SUBAPPLICATION GreenWhiteBackground3_AXSC (* Hintergrundfarbe (TRUE -> Grün, FALSE -> Weiß) für 3 Objekte (AX-Adapter) (Kompakt) *)
  (* Standard: 61499-2 *)
  (* Version 1.0, 2022-11-10, Franz Höpfinger, Meisterschulen am Ostbahnhof *)
  PACKAGE MyLib::sys;
  IMPORT isobus::UT::Q::const::IDs::ID_NULL;
  IMPORT isobus::UT::Q::types::s2ObjectIDs;
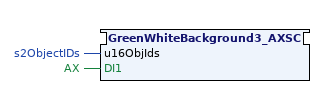
  VAR_INPUT
    u16ObjIds : isobus::UT::Q::types::s2ObjectIDs := (u16ObjId := ID_NULL, u16ObjIdA := ID_NULL); (* Object IDs *)
  END_VAR
  SOCKETS
    DI1 : adapter::types::unidirectional::AX; (* Selector *)
  END_SOCKETS
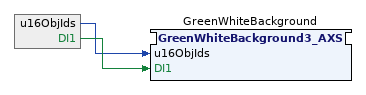
  SUBAPPS
    GreenWhiteBackground : MyLib::sys::GreenWhiteBackground3_AXS;
  END_SUBAPPS
  DATA_CONNECTIONS
    u16ObjIds TO GreenWhiteBackground.u16ObjIds;
  END_CONNECTIONS
  ADAPTER_CONNECTIONS
    DI1 TO GreenWhiteBackground.DI1;
  END_CONNECTIONS
END_SUBAPPLICATION
